KUKA KRL program: chk_w6_grp3_clo.src

&ACCESS RVO4
&COMMENT Check GRP AXOR Z3 CLOSE
DEF chk_w6_grp3_clo( )

; Check gripper axor CLOSE Z3.1
;//---- Start User-------

$TIMER[10] = 0
$TIMER_STOP[10] = FALSE

WAIT FOR (NOT $IN[497])
WAIT FOR ($IN[498])

$TIMER_STOP[10] = TRUE
$TIMER[10] = 0

;//---- End User---------
END
